TYPE ST_OutputStationHSJobDataOP11601 :
STRUCT
	{attribute 'OPC.UA.DA.Description' := 'Dynamic Tool'}
	{attribute 'OPC.UA.DA.StructuredType' := '1'}
	DynamicTool						: ARRAY [1..1] OF ToolX;

	{attribute 'OPC.UA.DA.Description' := 'Dynamic Material'}
	DynamicMaterial					: ARRAY [1..1] OF STRING(30);

	{attribute 'OPC.UA.DA.Description' := 'Temperature Target C°'}
	TemperatureTarget				: REAL;

	{attribute 'OPC.UA.DA.Description' := 'Temperature Max C°'}
	TemperatureMax					: REAL;
	
	{attribute 'OPC.UA.DA.Description' := 'Temperature Min C°'}
	TemperatureMin					: REAL;
	
	{attribute 'OPC.UA.DA.Description' := 'Time Max S'}
	TimeMax							: REAL;
	
	{attribute 'OPC.UA.DA.Description' := 'Time Min S'}
	TimeMin							: REAL;
	
	{attribute 'OPC.UA.DA.Description' := 'Steam Max'}
	SteamMax						: REAL;
	
	{attribute 'OPC.UA.DA.Description' := 'Steam Min'}
	SteamMin						: REAL;
	
	{attribute 'OPC.UA.DA.Description' := 'Air Max'}
	AirMax							: REAL;
	
	{attribute 'OPC.UA.DA.Description' := 'Air Min'}
	AirMin							: REAL;
	
	{attribute 'OPC.UA.DA.Description' := 'Profile'}
	Profile							: ARRAY [ 1..10] OF REAL;
	
END_STRUCT
END_TYPE

(* stored: Version 1.1.0.1, ProductVersion 3.1.4024.2
   DUT ST_OutputStationHSJobDataOP11601: Id {844bee34-5b8c-498d-b607-c68574daac8e} *)
